// TIA Portal project "Nastro con lavorazione HMI_lab" (V16)

(* hardware
DEVICE "HMI_1"  KTP700 Basic PN
   slot 0: "HMI_1"  KTP700 Basic PN  6AV2 123-2GB03-0AX0  16.0.0.0
   slot 1: "HMI_RT_1"  KTP700 Basic PN  6AV2 123-2GB03-0AX0  16.0.0.0
   slot 5: "HMI_1.IE_CP_1"  PROFINET Interface  16.0.0.0
      slot 1: "Interfaccia_1 PROFINET"  PROFINET Interface
         slot 1: "Porta_1"  Port
DEVICE "S7-1200 station_1"  S7-1200 Station
   slot 0: "Telaio di montaggio_0"  S7-1200 Rack  Rack  V1.0
   slot 1: "PLC_1"  CPU 1215C DC/DC/Rly  6ES7 215-1HG40-0XB0  V4.2
*)

// ===== PLC "PLC_1"  CPU 1215C DC/DC/Rly =====

VAR_GLOBAL   // PLC tag table "Tabella delle variabili standard"
   "Passo_0" AT %M0.0 : Bool;
   "Passo_1" AT %M0.1 : Bool;
   "Passo_2" AT %M0.2 : Bool;
   "Passo_3" AT %M0.3 : Bool;
   "Passo_4" AT %M0.4 : Bool;
   "BC_inizio" AT %I0.0 : Bool;
   "BC_fine" AT %I0.1 : Bool;
   "SQ_alto" AT %I0.2 : Bool;
   "SB_basso" AT %I0.3 : Bool;
   "Avanti nastro" AT %Q0.0 : Bool;
   "Indietro nastro" AT %Q0.1 : Bool;
   "Passo_5" AT %M0.5 : Bool;
   "Discesa lavorazione" AT %Q0.2 : Bool;
   "Salita lavorazione" AT %Q0.3 : Bool;
   "Clock_Byte" AT %MB10 : Byte;
   "Clock_10Hz" AT %M10.0 : Bool;
   "Clock_5Hz" AT %M10.1 : Bool;
   "Clock_2.5Hz" AT %M10.2 : Bool;
   "Clock_2Hz" AT %M10.3 : Bool;
   "Clock_1.25Hz" AT %M10.4 : Bool;
   "Clock_1Hz" AT %M10.5 : Bool;
   "Clock_0.625Hz" AT %M10.6 : Bool;
   "Clock_0.5Hz" AT %M10.7 : Bool;
END_VAR

DATA_BLOCK "Blocco_dati_HMI"   // DB1
{ S7_Optimized_Access := 'TRUE' }
VERSION : 0.1
   VAR
      jog_start : Bool;
      jog_BC_inizio : Bool;
      M_cicli : Bool;
      "movimento cilindretto" : Int;
      M_clock_veloce : Bool;
      M_clock_lento : Bool;
      "movimento lavorazione" : Int;
      jog_emergenza : Bool;
      jog_ripristino : Bool;
      M_tempo_lav : Bool;
      jog_BC_fine : Bool;
      jog_SQ_basso : Bool;
      jog_SQ_alto : Bool;
      preset_tempo_lav : Time;
      jog_carica_impostazioni : Bool;
      imposta_tempo_lav : Time;
      "lettura tempo_lav" : Time;
      "imposta numero di cicli" : Int;
      "lettura numero di cicli" : Int;
      preset_conteggio_cicli : Int;
      M_ripristino_cilindretto : Bool;
      M_ripristino_lav : Bool;
      Spia_BC_inizio : Bool;
      Spia_BC_fine : Bool;
      Spia_SQ_alto : Bool;
      "Spia _SQ_basso" : Bool;
      "Spia organi in movimento" : Bool;
      M_ripristino_lav_reale : Bool;
      M_ripristino_cilindro_reale_1 : Bool;
   END_VAR
BEGIN
END_DATA_BLOCK

// folder: System blocks/Program resources

DATA_BLOCK "Clock_lento"   // DB2
{ S7_Optimized_Access := 'TRUE' }
AUTHOR : Simatic
FAMILY : IEC
NAME : IEC_TMR
VERSION : 1.0
// stored: InstanceOfName IEC_TIMER
"IEC_TIMER"
BEGIN
END_DATA_BLOCK

DATA_BLOCK "Clock_veloce"   // DB3
{ S7_Optimized_Access := 'TRUE' }
AUTHOR : Simatic
FAMILY : IEC
NAME : IEC_TMR
VERSION : 1.0
// stored: InstanceOfName IEC_TIMER
"IEC_TIMER"
BEGIN
END_DATA_BLOCK

DATA_BLOCK "Tempo_lav"   // DB4
{ S7_Optimized_Access := 'TRUE' }
AUTHOR : Simatic
FAMILY : IEC
NAME : IEC_TMR
VERSION : 1.0
// stored: InstanceOfName IEC_TIMER
"IEC_TIMER"
BEGIN
END_DATA_BLOCK

DATA_BLOCK "Conteggio cicli"   // DB5
{ S7_Optimized_Access := 'TRUE' }
AUTHOR : Simatic
FAMILY : IEC
NAME : CNTR
VERSION : 1.0
// stored: InstanceOfName IEC_COUNTER
"IEC_COUNTER"
BEGIN
END_DATA_BLOCK

// folder: (top level)

FUNCTION "Ripristino" : Void   // FC1, LAD
{ S7_Optimized_Access := 'TRUE' }
VERSION : 0.1
BEGIN

REGION Network 1
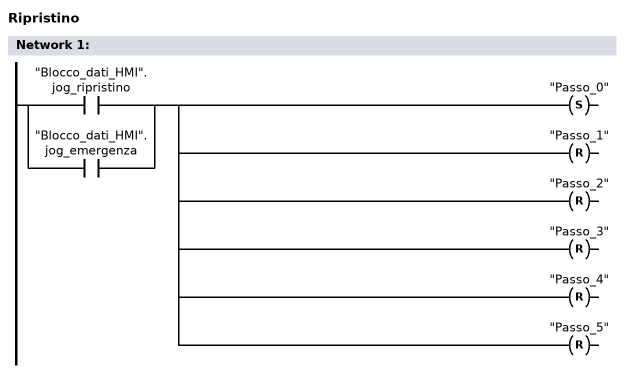
   RUNG wire#powerrail
      Contact( "Blocco_dati_HMI".jog_ripristino )
      wire#w1
      S_Coil( "Passo_0" )
   END_RUNG
   RUNG wire#powerrail
      Contact( "Blocco_dati_HMI".jog_emergenza )
   END_RUNG wire#w1
   RUNG wire#w1
      R_Coil( "Passo_1" )
   END_RUNG
   RUNG wire#w1
      R_Coil( "Passo_2" )
   END_RUNG
   RUNG wire#w1
      R_Coil( "Passo_3" )
   END_RUNG
   RUNG wire#w1
      R_Coil( "Passo_4" )
   END_RUNG
   RUNG wire#w1
      R_Coil( "Passo_5" )
   END_RUNG
   // the same network as SCL:
   IF "Blocco_dati_HMI".jog_ripristino OR "Blocco_dati_HMI".jog_emergenza THEN
       "Passo_0" := TRUE;
       "Passo_1" := FALSE;
       "Passo_2" := FALSE;
       "Passo_3" := FALSE;
       "Passo_4" := FALSE;
       "Passo_5" := FALSE;
   END_IF;
END_REGION
END_FUNCTION

FUNCTION "Struttura dei passi" : Void   // FC2, LAD
{ S7_Optimized_Access := 'TRUE' }
VERSION : 0.1
   VAR_TEMP   // added for the SCL form of the ladder/FBD networks
      _w1 : Bool;
   END_VAR
BEGIN

REGION Network 1
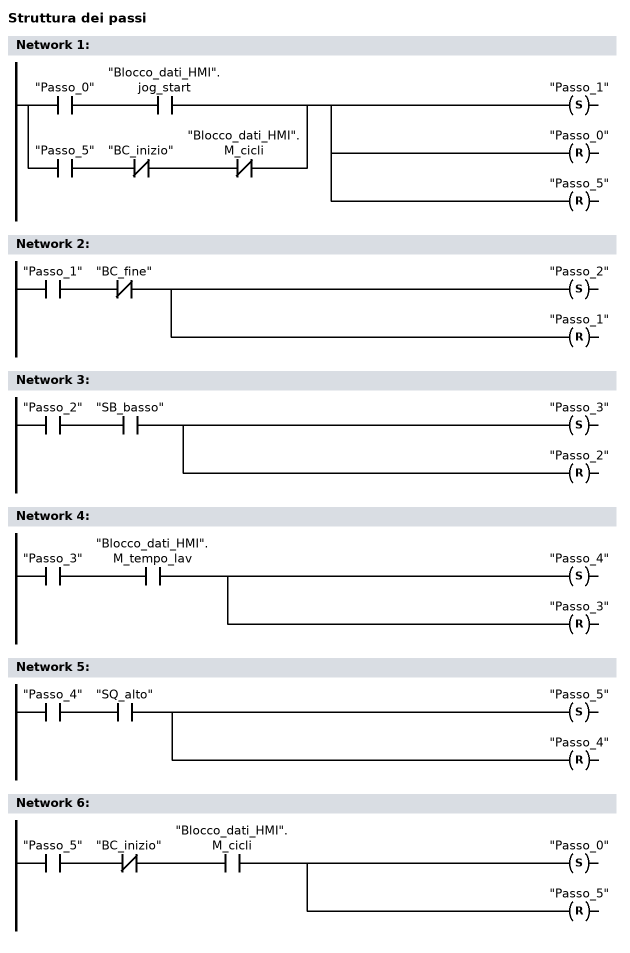
   RUNG wire#powerrail
      Contact( "Passo_0" )
      Contact( "Blocco_dati_HMI".jog_start )
      wire#w1
      S_Coil( "Passo_1" )
   END_RUNG
   RUNG wire#powerrail
      Contact( "Passo_5" )
      I_Contact( "BC_inizio" )
      I_Contact( "Blocco_dati_HMI".M_cicli )
   END_RUNG wire#w1
   RUNG wire#w1
      R_Coil( "Passo_0" )
   END_RUNG
   RUNG wire#w1
      R_Coil( "Passo_5" )
   END_RUNG
   // the same network as SCL:
   IF ("Passo_0" AND "Blocco_dati_HMI".jog_start) OR ("Passo_5" AND NOT "BC_inizio" AND NOT "Blocco_dati_HMI".M_cicli) THEN
       "Passo_1" := TRUE;
   END_IF;
   #_w1 := ("Passo_0" AND "Blocco_dati_HMI".jog_start) OR ("Passo_5" AND NOT "BC_inizio" AND NOT "Blocco_dati_HMI".M_cicli);
   IF #_w1 THEN
       "Passo_0" := FALSE;
       "Passo_5" := FALSE;
   END_IF;
END_REGION

REGION Network 2
   RUNG wire#powerrail
      Contact( "Passo_1" )
      I_Contact( "BC_fine" )
      wire#w1
      S_Coil( "Passo_2" )
   END_RUNG
   RUNG wire#w1
      R_Coil( "Passo_1" )
   END_RUNG
   // the same network as SCL:
   IF "Passo_1" AND NOT "BC_fine" THEN
       "Passo_2" := TRUE;
       "Passo_1" := FALSE;
   END_IF;
END_REGION

REGION Network 3
   RUNG wire#powerrail
      Contact( "Passo_2" )
      Contact( "SB_basso" )
      wire#w1
      S_Coil( "Passo_3" )
   END_RUNG
   RUNG wire#w1
      R_Coil( "Passo_2" )
   END_RUNG
   // the same network as SCL:
   IF "Passo_2" AND "SB_basso" THEN
       "Passo_3" := TRUE;
       "Passo_2" := FALSE;
   END_IF;
END_REGION

REGION Network 4
   RUNG wire#powerrail
      Contact( "Passo_3" )
      Contact( "Blocco_dati_HMI".M_tempo_lav )
      wire#w1
      S_Coil( "Passo_4" )
   END_RUNG
   RUNG wire#w1
      R_Coil( "Passo_3" )
   END_RUNG
   // the same network as SCL:
   IF "Passo_3" AND "Blocco_dati_HMI".M_tempo_lav THEN
       "Passo_4" := TRUE;
       "Passo_3" := FALSE;
   END_IF;
END_REGION

REGION Network 5
   RUNG wire#powerrail
      Contact( "Passo_4" )
      Contact( "SQ_alto" )
      wire#w1
      S_Coil( "Passo_5" )
   END_RUNG
   RUNG wire#w1
      R_Coil( "Passo_4" )
   END_RUNG
   // the same network as SCL:
   IF "Passo_4" AND "SQ_alto" THEN
       "Passo_5" := TRUE;
       "Passo_4" := FALSE;
   END_IF;
END_REGION

REGION Network 6
   RUNG wire#powerrail
      Contact( "Passo_5" )
      I_Contact( "BC_inizio" )
      Contact( "Blocco_dati_HMI".M_cicli )
      wire#w1
      S_Coil( "Passo_0" )
   END_RUNG
   RUNG wire#w1
      R_Coil( "Passo_5" )
   END_RUNG
   // the same network as SCL:
   IF "Passo_5" AND NOT "BC_inizio" AND "Blocco_dati_HMI".M_cicli THEN
       "Passo_0" := TRUE;
       "Passo_5" := FALSE;
   END_IF;
END_REGION
END_FUNCTION

FUNCTION "Attivazione delle uscite" : Void   // FC3, LAD
{ S7_Optimized_Access := 'TRUE' }
VERSION : 0.1
BEGIN

REGION Network 1
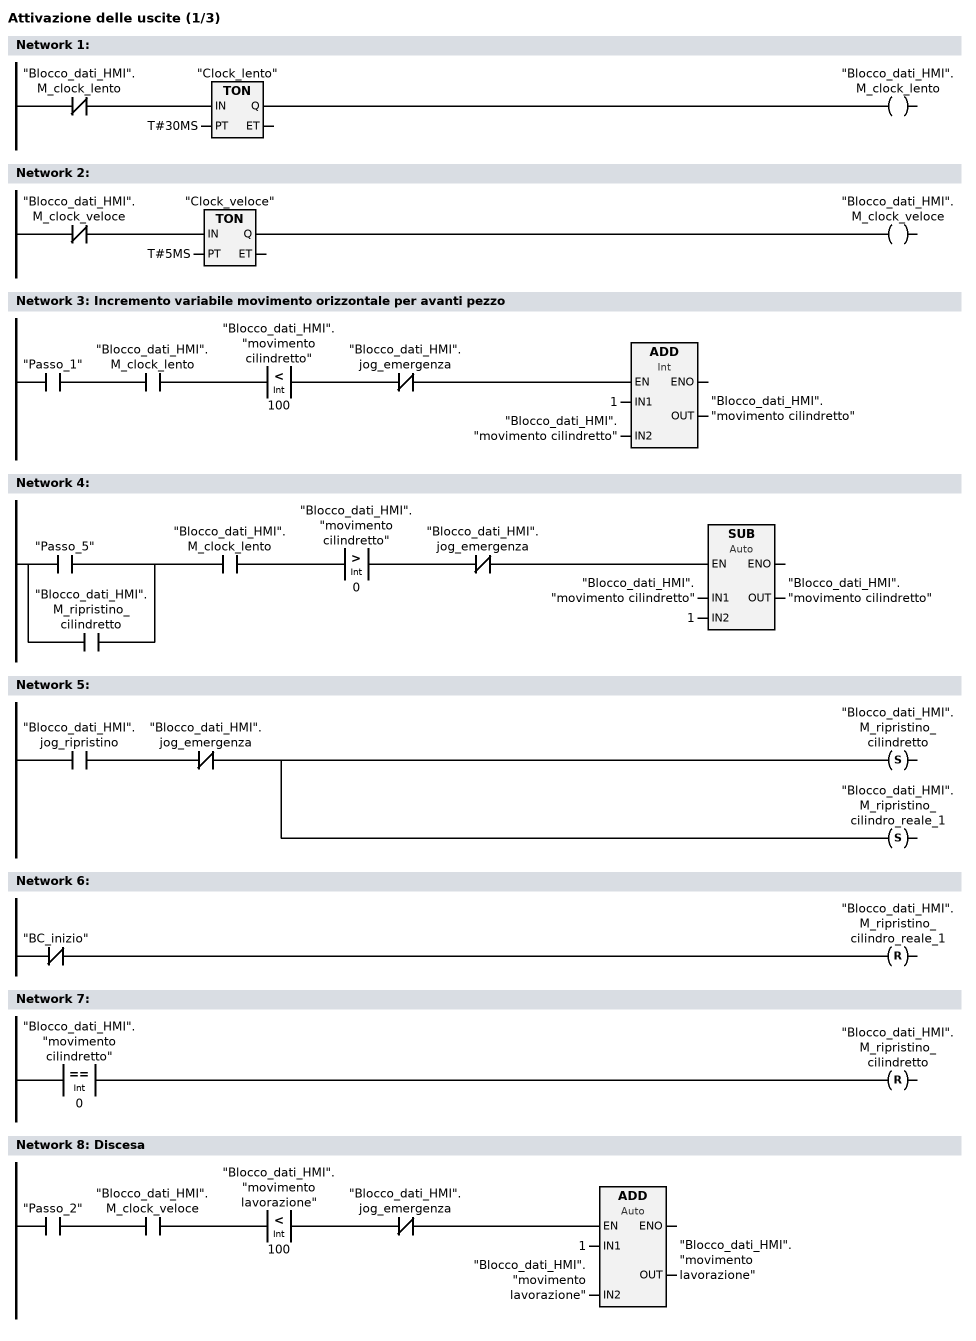
   "Clock_lento".TON(IN := NOT "Blocco_dati_HMI".M_clock_lento, PT := T#30MS);
   "Blocco_dati_HMI".M_clock_lento := "Clock_lento".Q;
END_REGION

REGION Network 2
   "Clock_veloce".TON(IN := NOT "Blocco_dati_HMI".M_clock_veloce, PT := T#5MS);
   "Blocco_dati_HMI".M_clock_veloce := "Clock_veloce".Q;
END_REGION

REGION Network 3: Incremento variabile movimento orizzontale per avanti pezzo
   RUNG wire#powerrail
      Contact( "Passo_1" )
      Contact( "Blocco_dati_HMI".M_clock_lento )
      { S7_Templates := "SrcType := Int" } LT_Contact(in1 := "Blocco_dati_HMI"."movimento cilindretto", in2 := 100)
      I_Contact( "Blocco_dati_HMI".jog_emergenza )
      { S7_Templates := "SrcType := Int" } Add(in1 := 1, in2 := "Blocco_dati_HMI"."movimento cilindretto", out => "Blocco_dati_HMI"."movimento cilindretto")
   END_RUNG
   // the same network as SCL:
   IF "Passo_1" AND "Blocco_dati_HMI".M_clock_lento AND ("Blocco_dati_HMI"."movimento cilindretto" < 100) AND NOT "Blocco_dati_HMI".jog_emergenza THEN
       "Blocco_dati_HMI"."movimento cilindretto" := 1 + "Blocco_dati_HMI"."movimento cilindretto";
   END_IF;
END_REGION

REGION Network 4
   RUNG wire#powerrail
      Contact( "Passo_5" )
      wire#w1
      Contact( "Blocco_dati_HMI".M_clock_lento )
      { S7_Templates := "SrcType := Int" } GT_Contact(in1 := "Blocco_dati_HMI"."movimento cilindretto", in2 := 0)
      I_Contact( "Blocco_dati_HMI".jog_emergenza )
      Sub(in1 := "Blocco_dati_HMI"."movimento cilindretto", in2 := 1, out => "Blocco_dati_HMI"."movimento cilindretto")
   END_RUNG
   RUNG wire#powerrail
      Contact( "Blocco_dati_HMI".M_ripristino_cilindretto )
   END_RUNG wire#w1
   // the same network as SCL:
   IF ("Passo_5" OR "Blocco_dati_HMI".M_ripristino_cilindretto) AND "Blocco_dati_HMI".M_clock_lento AND ("Blocco_dati_HMI"."movimento cilindretto" > 0) AND NOT "Blocco_dati_HMI".jog_emergenza THEN
       "Blocco_dati_HMI"."movimento cilindretto" := "Blocco_dati_HMI"."movimento cilindretto" - 1;
   END_IF;
END_REGION

REGION Network 5
   RUNG wire#powerrail
      Contact( "Blocco_dati_HMI".jog_ripristino )
      I_Contact( "Blocco_dati_HMI".jog_emergenza )
      wire#w1
      S_Coil( "Blocco_dati_HMI".M_ripristino_cilindretto )
   END_RUNG
   RUNG wire#w1
      S_Coil( "Blocco_dati_HMI".M_ripristino_cilindro_reale_1 )
   END_RUNG
   // the same network as SCL:
   IF "Blocco_dati_HMI".jog_ripristino AND NOT "Blocco_dati_HMI".jog_emergenza THEN
       "Blocco_dati_HMI".M_ripristino_cilindretto := TRUE;
       "Blocco_dati_HMI".M_ripristino_cilindro_reale_1 := TRUE;
   END_IF;
END_REGION

REGION Network 6
   RUNG wire#powerrail
      I_Contact( "BC_inizio" )
      R_Coil( "Blocco_dati_HMI".M_ripristino_cilindro_reale_1 )
   END_RUNG
   // the same network as SCL:
   IF NOT "BC_inizio" THEN "Blocco_dati_HMI".M_ripristino_cilindro_reale_1 := FALSE; END_IF;
END_REGION

REGION Network 7
   RUNG wire#powerrail
      { S7_Templates := "SrcType := Int" } EQ_Contact(in1 := "Blocco_dati_HMI"."movimento cilindretto", in2 := 0)
      R_Coil( "Blocco_dati_HMI".M_ripristino_cilindretto )
   END_RUNG
   // the same network as SCL:
   IF "Blocco_dati_HMI"."movimento cilindretto" = 0 THEN
       "Blocco_dati_HMI".M_ripristino_cilindretto := FALSE;
   END_IF;
END_REGION

REGION Network 8: Discesa
   RUNG wire#powerrail
      Contact( "Passo_2" )
      Contact( "Blocco_dati_HMI".M_clock_veloce )
      { S7_Templates := "SrcType := Int" } LT_Contact(in1 := "Blocco_dati_HMI"."movimento lavorazione", in2 := 100)
      I_Contact( "Blocco_dati_HMI".jog_emergenza )
      Add(in1 := 1, in2 := "Blocco_dati_HMI"."movimento lavorazione", out => "Blocco_dati_HMI"."movimento lavorazione")
   END_RUNG
   // the same network as SCL:
   IF "Passo_2" AND "Blocco_dati_HMI".M_clock_veloce AND ("Blocco_dati_HMI"."movimento lavorazione" < 100) AND NOT "Blocco_dati_HMI".jog_emergenza THEN
       "Blocco_dati_HMI"."movimento lavorazione" := 1 + "Blocco_dati_HMI"."movimento lavorazione";
   END_IF;
END_REGION

REGION Network 9: salita
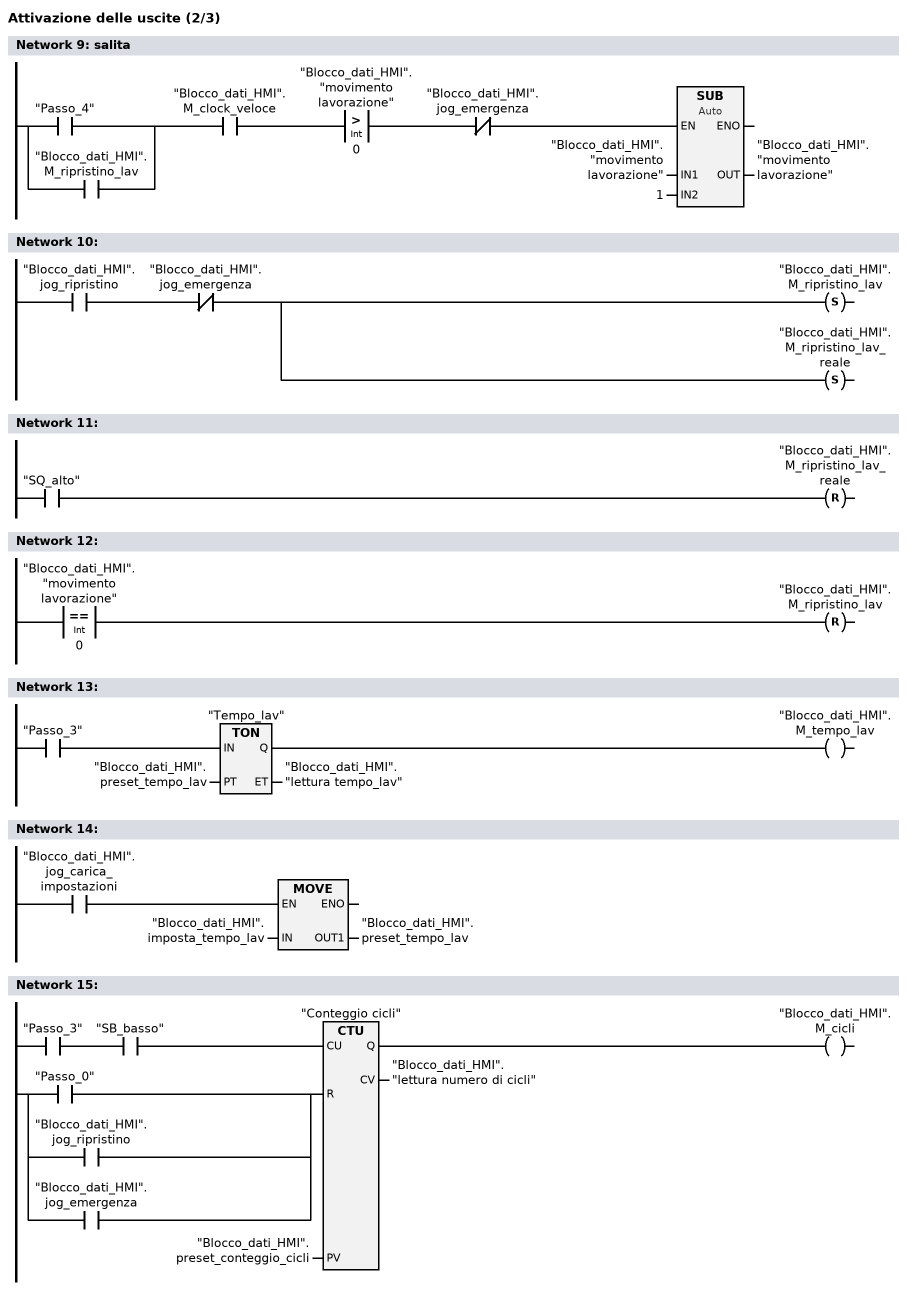
   RUNG wire#powerrail
      Contact( "Passo_4" )
      wire#w1
      Contact( "Blocco_dati_HMI".M_clock_veloce )
      { S7_Templates := "SrcType := Int" } GT_Contact(in1 := "Blocco_dati_HMI"."movimento lavorazione", in2 := 0)
      I_Contact( "Blocco_dati_HMI".jog_emergenza )
      Sub(in1 := "Blocco_dati_HMI"."movimento lavorazione", in2 := 1, out => "Blocco_dati_HMI"."movimento lavorazione")
   END_RUNG
   RUNG wire#powerrail
      Contact( "Blocco_dati_HMI".M_ripristino_lav )
   END_RUNG wire#w1
   // the same network as SCL:
   IF ("Passo_4" OR "Blocco_dati_HMI".M_ripristino_lav) AND "Blocco_dati_HMI".M_clock_veloce AND ("Blocco_dati_HMI"."movimento lavorazione" > 0) AND NOT "Blocco_dati_HMI".jog_emergenza THEN
       "Blocco_dati_HMI"."movimento lavorazione" := "Blocco_dati_HMI"."movimento lavorazione" - 1;
   END_IF;
END_REGION

REGION Network 10
   RUNG wire#powerrail
      Contact( "Blocco_dati_HMI".jog_ripristino )
      I_Contact( "Blocco_dati_HMI".jog_emergenza )
      wire#w1
      S_Coil( "Blocco_dati_HMI".M_ripristino_lav )
   END_RUNG
   RUNG wire#w1
      S_Coil( "Blocco_dati_HMI".M_ripristino_lav_reale )
   END_RUNG
   // the same network as SCL:
   IF "Blocco_dati_HMI".jog_ripristino AND NOT "Blocco_dati_HMI".jog_emergenza THEN
       "Blocco_dati_HMI".M_ripristino_lav := TRUE;
       "Blocco_dati_HMI".M_ripristino_lav_reale := TRUE;
   END_IF;
END_REGION

REGION Network 11
   RUNG wire#powerrail
      Contact( "SQ_alto" )
      R_Coil( "Blocco_dati_HMI".M_ripristino_lav_reale )
   END_RUNG
   // the same network as SCL:
   IF "SQ_alto" THEN "Blocco_dati_HMI".M_ripristino_lav_reale := FALSE; END_IF;
END_REGION

REGION Network 12
   RUNG wire#powerrail
      { S7_Templates := "SrcType := Int" } EQ_Contact(in1 := "Blocco_dati_HMI"."movimento lavorazione", in2 := 0)
      R_Coil( "Blocco_dati_HMI".M_ripristino_lav )
   END_RUNG
   // the same network as SCL:
   IF "Blocco_dati_HMI"."movimento lavorazione" = 0 THEN "Blocco_dati_HMI".M_ripristino_lav := FALSE; END_IF;
END_REGION

REGION Network 13
   "Tempo_lav".TON(IN := "Passo_3",
                   PT := "Blocco_dati_HMI".preset_tempo_lav,
                   ET => "Blocco_dati_HMI"."lettura tempo_lav");
   "Blocco_dati_HMI".M_tempo_lav := "Tempo_lav".Q;
END_REGION

REGION Network 14
   RUNG wire#powerrail
      Contact( "Blocco_dati_HMI".jog_carica_impostazioni )
      Move(in := "Blocco_dati_HMI".imposta_tempo_lav, out1 => "Blocco_dati_HMI".preset_tempo_lav)
   END_RUNG
   // the same network as SCL:
   IF "Blocco_dati_HMI".jog_carica_impostazioni THEN
       "Blocco_dati_HMI".preset_tempo_lav := "Blocco_dati_HMI".imposta_tempo_lav;
   END_IF;
END_REGION

REGION Network 15
   "Conteggio cicli".CTU(CU := "Passo_3" AND "SB_basso",
                         R := "Passo_0" OR "Blocco_dati_HMI".jog_ripristino OR "Blocco_dati_HMI".jog_emergenza,
                         PV := "Blocco_dati_HMI".preset_conteggio_cicli,
                         CV => "Blocco_dati_HMI"."lettura numero di cicli");
   "Blocco_dati_HMI".M_cicli := "Conteggio cicli".Q;
END_REGION

REGION Network 16
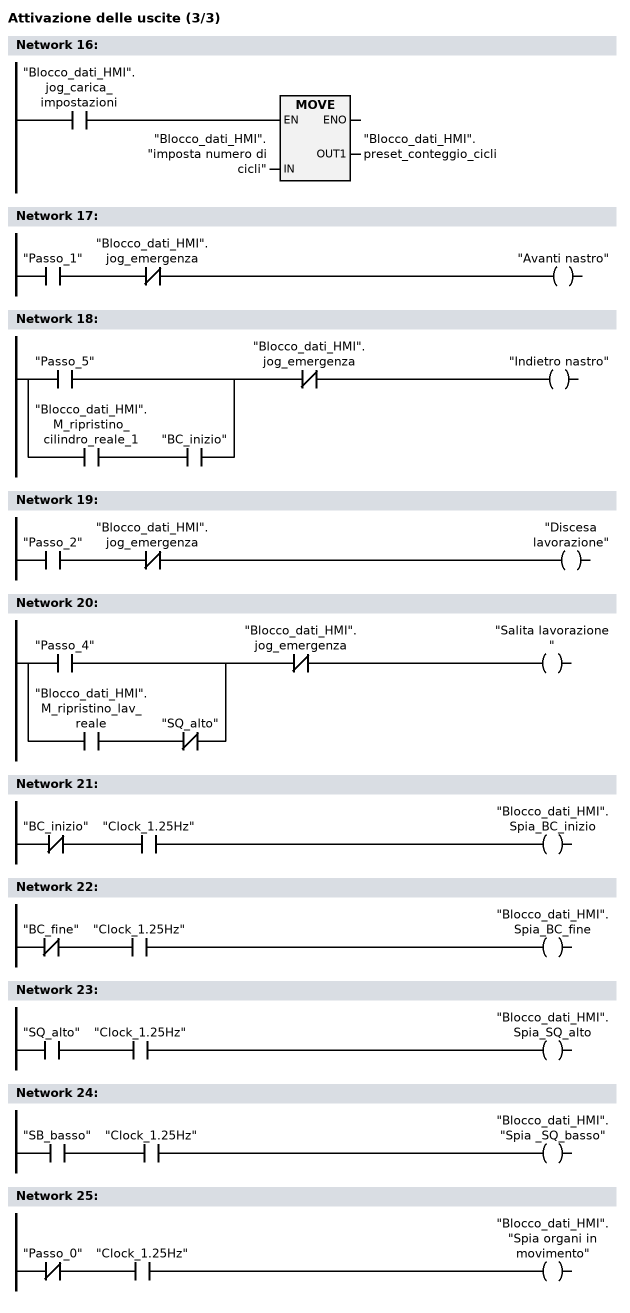
   RUNG wire#powerrail
      Contact( "Blocco_dati_HMI".jog_carica_impostazioni )
      Move(in := "Blocco_dati_HMI"."imposta numero di cicli", out1 => "Blocco_dati_HMI".preset_conteggio_cicli)
   END_RUNG
   // the same network as SCL:
   IF "Blocco_dati_HMI".jog_carica_impostazioni THEN
       "Blocco_dati_HMI".preset_conteggio_cicli := "Blocco_dati_HMI"."imposta numero di cicli";
   END_IF;
END_REGION

REGION Network 17
   RUNG wire#powerrail
      Contact( "Passo_1" )
      I_Contact( "Blocco_dati_HMI".jog_emergenza )
      Coil( "Avanti nastro" )
   END_RUNG
   // the same network as SCL:
   "Avanti nastro" := "Passo_1" AND NOT "Blocco_dati_HMI".jog_emergenza;
END_REGION

REGION Network 18
   RUNG wire#powerrail
      Contact( "Passo_5" )
      wire#w1
      I_Contact( "Blocco_dati_HMI".jog_emergenza )
      Coil( "Indietro nastro" )
   END_RUNG
   RUNG wire#powerrail
      Contact( "Blocco_dati_HMI".M_ripristino_cilindro_reale_1 )
      Contact( "BC_inizio" )
   END_RUNG wire#w1
   // the same network as SCL:
   "Indietro nastro" := ("Passo_5" OR ("Blocco_dati_HMI".M_ripristino_cilindro_reale_1 AND "BC_inizio")) AND NOT "Blocco_dati_HMI".jog_emergenza;
END_REGION

REGION Network 19
   RUNG wire#powerrail
      Contact( "Passo_2" )
      I_Contact( "Blocco_dati_HMI".jog_emergenza )
      Coil( "Discesa lavorazione" )
   END_RUNG
   // the same network as SCL:
   "Discesa lavorazione" := "Passo_2" AND NOT "Blocco_dati_HMI".jog_emergenza;
END_REGION

REGION Network 20
   RUNG wire#powerrail
      Contact( "Passo_4" )
      wire#w1
      I_Contact( "Blocco_dati_HMI".jog_emergenza )
      Coil( "Salita lavorazione" )
   END_RUNG
   RUNG wire#powerrail
      Contact( "Blocco_dati_HMI".M_ripristino_lav_reale )
      I_Contact( "SQ_alto" )
   END_RUNG wire#w1
   // the same network as SCL:
   "Salita lavorazione" := ("Passo_4" OR ("Blocco_dati_HMI".M_ripristino_lav_reale AND NOT "SQ_alto")) AND NOT "Blocco_dati_HMI".jog_emergenza;
END_REGION

REGION Network 21
   RUNG wire#powerrail
      I_Contact( "BC_inizio" )
      Contact( "Clock_1.25Hz" )
      Coil( "Blocco_dati_HMI".Spia_BC_inizio )
   END_RUNG
   // the same network as SCL:
   "Blocco_dati_HMI".Spia_BC_inizio := NOT "BC_inizio" AND "Clock_1.25Hz";
END_REGION

REGION Network 22
   RUNG wire#powerrail
      I_Contact( "BC_fine" )
      Contact( "Clock_1.25Hz" )
      Coil( "Blocco_dati_HMI".Spia_BC_fine )
   END_RUNG
   // the same network as SCL:
   "Blocco_dati_HMI".Spia_BC_fine := NOT "BC_fine" AND "Clock_1.25Hz";
END_REGION

REGION Network 23
   RUNG wire#powerrail
      Contact( "SQ_alto" )
      Contact( "Clock_1.25Hz" )
      Coil( "Blocco_dati_HMI".Spia_SQ_alto )
   END_RUNG
   // the same network as SCL:
   "Blocco_dati_HMI".Spia_SQ_alto := "SQ_alto" AND "Clock_1.25Hz";
END_REGION

REGION Network 24
   RUNG wire#powerrail
      Contact( "SB_basso" )
      Contact( "Clock_1.25Hz" )
      Coil( "Blocco_dati_HMI"."Spia _SQ_basso" )
   END_RUNG
   // the same network as SCL:
   "Blocco_dati_HMI"."Spia _SQ_basso" := "SB_basso" AND "Clock_1.25Hz";
END_REGION

REGION Network 25
   RUNG wire#powerrail
      I_Contact( "Passo_0" )
      Contact( "Clock_1.25Hz" )
      Coil( "Blocco_dati_HMI"."Spia organi in movimento" )
   END_RUNG
   // the same network as SCL:
   "Blocco_dati_HMI"."Spia organi in movimento" := NOT "Passo_0" AND "Clock_1.25Hz";
END_REGION
END_FUNCTION

ORGANIZATION_BLOCK "Main"   // OB1, LAD, ProgramCycle
TITLE = "Main Program Sweep (Cycle)"
{ S7_Optimized_Access := 'TRUE' }
VERSION : 0.1
   VAR_INPUT
      Initial_Call : Bool;   // Initial call of this OB
      Remanence : Bool;   // =True, if remanent data are available
   END_VAR
BEGIN

REGION Network 1
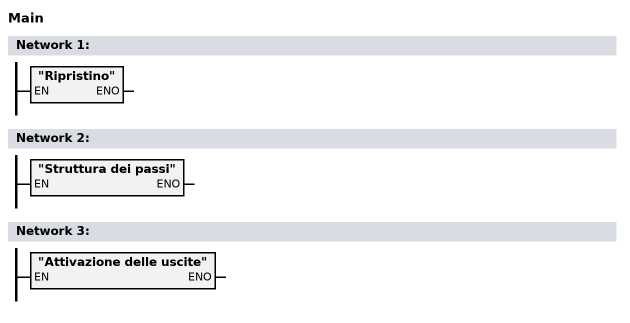
   RUNG wire#powerrail
      "Ripristino"()
   END_RUNG
   // the same network as SCL:
   "Ripristino"();
END_REGION

REGION Network 2
   RUNG wire#powerrail
      "Struttura dei passi"()
   END_RUNG
   // the same network as SCL:
   "Struttura dei passi"();
END_REGION

REGION Network 3
   RUNG wire#powerrail
      "Attivazione delle uscite"()
   END_RUNG
   // the same network as SCL:
   "Attivazione delle uscite"();
END_REGION
END_ORGANIZATION_BLOCK

(* ===== HMI "HMI_RT_1" =====
system functions are stored by id; their names below are inferred from use
connection "HMI_Collegamento_1": ETHERNET, SMART_S7_1200_OMS

HMI tags "Tabella delle variabili standard"
   "Blocco_dati_HMI_jog_emergenza" : Bool = PLC Blocco_dati_HMI.jog_emergenza, 100 ms
   "Blocco_dati_HMI_jog_ripristino" : Bool = PLC Blocco_dati_HMI.jog_ripristino, 100 ms
   "Blocco_dati_HMI_jog_start" : Bool = PLC Blocco_dati_HMI.jog_start, 100 ms
   "Blocco_dati_HMI_imposta_tempo_lav" : Time = PLC Blocco_dati_HMI.imposta_tempo_lav, 100 ms
   "Blocco_dati_HMI_preset_tempo_lav" : Time = PLC Blocco_dati_HMI.preset_tempo_lav, 100 ms
   "Blocco_dati_HMI_lettura tempo_lav" : Time = PLC Blocco_dati_HMI."lettura tempo_lav", 100 ms
   "Blocco_dati_HMI_imposta numero di cicli" : Int = PLC Blocco_dati_HMI."imposta numero di cicli", 100 ms
   "Blocco_dati_HMI_preset_conteggio_cicli" : Int = PLC Blocco_dati_HMI.preset_conteggio_cicli, 100 ms
   "Blocco_dati_HMI_lettura numero di cicli" : Int = PLC Blocco_dati_HMI."lettura numero di cicli", 100 ms
   "Blocco_dati_HMI_jog_carica_impostazioni" : Bool = PLC Blocco_dati_HMI.jog_carica_impostazioni, 100 ms
   "Blocco_dati_HMI_jog_BC_inizio" : Bool = PLC Blocco_dati_HMI.jog_BC_inizio, 100 ms
   "Blocco_dati_HMI_jog_BC_fine" : Bool = PLC Blocco_dati_HMI.jog_BC_fine, 100 ms
   "Blocco_dati_HMI_jog_SQ_basso" : Bool = PLC Blocco_dati_HMI.jog_SQ_basso, 100 ms
   "Blocco_dati_HMI_jog_SQ_alto" : Bool = PLC Blocco_dati_HMI.jog_SQ_alto, 100 ms
   "Blocco_dati_HMI_movimento cilindretto" : Int = PLC Blocco_dati_HMI."movimento cilindretto", 100 ms
   "Blocco_dati_HMI_movimento lavorazione" : Int = PLC Blocco_dati_HMI."movimento lavorazione", 100 ms
   "Blocco_dati_HMI_Spia organi in movimento" : Bool = PLC Blocco_dati_HMI."Spia organi in movimento", 100 ms
   "Blocco_dati_HMI_Spia_SQ_alto" : Bool = PLC Blocco_dati_HMI.Spia_SQ_alto, 100 ms
   "Blocco_dati_HMI_Spia _SQ_basso" : Bool = PLC Blocco_dati_HMI."Spia _SQ_basso", 100 ms
   "Blocco_dati_HMI_Spia_BC_fine" : Bool = PLC Blocco_dati_HMI.Spia_BC_fine, 100 ms
   "Blocco_dati_HMI_Spia_BC_inizio" : Bool = PLC Blocco_dati_HMI.Spia_BC_inizio, 100 ms

screen "Pagina_1" 800x480
   Softkey "Softkey_F1" at 0,0 size 0x0
      on KeyDown: ActivateScreen("Pagina_1", 0)
   Softkey "Softkey_F2" at 0,0 size 0x0
      on KeyDown: ActivateScreen("Pagina_2", 0)

screen "Pagina_2" 800x480
   Softkey "Softkey_F1" at 0,0 size 0x0
      on KeyDown: ActivateScreen("Pagina_1", 0)
   Softkey "Softkey_F2" at 0,0 size 0x0
      on KeyDown: ActivateScreen("Pagina_2", 0)
   Rectangle "Rettangolo_2" at 526,291 size 46x43
      HorizontalMovement <- "Blocco_dati_HMI_movimento cilindretto"
   Switch "Pushbutton_Emergency" at 53,43 size 80x80; CaptionText 'Switch'; TextOff '0'; TextOn '1'; PictureOff "Pushbutton_Emergency_Off_256c"; PictureOn "Pushbutton_Emergency_On_256c"
      on SwitchOn: SetBit("Blocco_dati_HMI_jog_emergenza")
      on SwitchOff: ResetBit("Blocco_dati_HMI_jog_emergenza")
   Button "FB_Home_Round" at 211,48 size 50x50; TextOff 'Text'; PictureOn "FB_Home_Round_Pressed_256c"; PictureOff "FB_Home_Round_Released_256c"
      on Press: SetBit("Blocco_dati_HMI_jog_ripristino")
      on Release: ResetBit("Blocco_dati_HMI_jog_ripristino")
   Button "FB_Right_Round" at 318,48 size 50x50; TextOff 'Text'; PictureOn "FB_Right_Round_Pressed_256c"; PictureOff "FB_Right_Round_Released_256c"
      on Press: SetBit("Blocco_dati_HMI_jog_start")
      on Release: ResetBit("Blocco_dati_HMI_jog_start")
   IOField "Campo I/O_1" at 47,240 size 58x32; FormatPattern 9999
      ProcessValue <- "Blocco_dati_HMI_imposta_tempo_lav"
   IOField "Campo I/O_2" at 47,403 size 58x32; FormatPattern 9999
      ProcessValue <- "Blocco_dati_HMI_imposta numero di cicli"
   IOField "Campo I/O_3" at 183,240 size 58x32; FormatPattern 9999
      ProcessValue <- "Blocco_dati_HMI_preset_tempo_lav"
   IOField "Campo I/O_4" at 183,403 size 58x32; FormatPattern 9999
      ProcessValue <- "Blocco_dati_HMI_preset_conteggio_cicli"
   IOField "Campo I/O_5" at 321,240 size 58x32; FormatPattern 9999
      ProcessValue <- "Blocco_dati_HMI_lettura tempo_lav"
   IOField "Campo I/O_6" at 320,402 size 58x32; FormatPattern 9999
      ProcessValue <- "Blocco_dati_HMI_lettura numero di cicli"
   Button "FB_Plus_Round" at 116,310 size 50x50; TextOff 'Text'; PictureOn "FB_Plus_Round_Pressed_256c"; PictureOff "FB_Plus_Round_Released_256c"
      on Press: SetBit("Blocco_dati_HMI_jog_carica_impostazioni")
      on Release: ResetBit("Blocco_dati_HMI_jog_carica_impostazioni")
   TextField "Casella di testo_1" at 53,19 size 76x20; Text 'Emergenza'
   TextField "Casella di testo_2" at 212,19 size 41x20; Text 'Home'
   TextField "Casella di testo_3" at 488,48 size 65x20; Text 'Macchina'
   TextField "Casella di testo_5" at 42,201 size 87x20; Text 'Digita tempo'
   TextField "Casella di testo_6" at 42,216 size 80x20; Text 'lavorazione'
   TextField "Casella di testo_4" at 183,201 size 47x20; Text 'Tempo'
   TextField "Casella di testo_7" at 183,216 size 80x20; Text 'lavorazione'
   TextField "Casella di testo_8" at 316,201 size 68x20; Text 'Visualizza'
   TextField "Casella di testo_9" at 316,216 size 88x20; Text 'tempo di lav.'
   TextField "Casella di testo_10" at 103,275 size 45x20; Text 'Carica'
   TextField "Casella di testo_11" at 103,290 size 85x20; Text 'impostazioni'
   TextField "Casella di testo_12" at 42,367 size 95x20; Text 'Digita numero'
   TextField "Casella di testo_13" at 42,382 size 43x20; Text 'di cicli'
   TextField "Casella di testo_14" at 184,368 size 58x20; Text 'Numero'
   TextField "Casella di testo_15" at 184,383 size 43x20; Text 'di cicli'
   TextField "Casella di testo_16" at 321,367 size 68x20; Text 'Visualizza'
   TextField "Casella di testo_17" at 321,382 size 96x20; Text 'numero di cicli'
   TextField "Casella di testo_18" at 727,60 size 49x17; Text 'SQ_alto'
   TextField "Casella di testo_19" at 725,237 size 60x17; Text 'SQ_basso'
   TextField "Casella di testo_20" at 498,384 size 55x17; Text 'BC_inizio'
   TextField "Casella di testo_21" at 668,383 size 47x17; Text 'BC_fine'
   TextField "Casella di testo_22" at 487,61 size 91x20; Text 'in movimento'
   TextField "Casella di testo_23" at 316,23 size 39x20; Text 'Start'
   Switch "Interruttore_1" at 503,363 size 45x21; CaptionText 'Switch'; TextOff 'OFF'; TextOn 'ON'
      on SwitchOn: SetBit("Blocco_dati_HMI_jog_BC_inizio")
      on SwitchOff: ResetBit("Blocco_dati_HMI_jog_BC_inizio")
   Switch "Interruttore_2" at 674,362 size 45x21; TextOn 'ON'; CaptionText 'Switch'; TextOff 'OFF'
      on SwitchOn: SetBit("Blocco_dati_HMI_jog_BC_fine")
      on SwitchOff: ResetBit("Blocco_dati_HMI_jog_BC_fine")
   Switch "Interruttore_3" at 727,81 size 45x21; TextOn 'ON'; CaptionText 'Switch'; TextOff 'OFF'
      on SwitchOn: SetBit("Blocco_dati_HMI_jog_SQ_alto")
      on SwitchOff: ResetBit("Blocco_dati_HMI_jog_SQ_alto")
   Switch "Interruttore_4" at 728,259 size 45x21; TextOn 'ON'; CaptionText 'Switch'; TextOff 'OFF'
      on SwitchOn: SetBit("Blocco_dati_HMI_jog_SQ_basso")
      on SwitchOff: ResetBit("Blocco_dati_HMI_jog_SQ_basso")
   GraphicIOField "PlotLight_Round_R" at 499,77 size 50x50; PictureOn "PilotLight_Round_R_On_256c"; PictureOff "PilotLight_Round_R_Off_256c"
      ProcessValue <- "Blocco_dati_HMI_Spia organi in movimento"
   GraphicIOField "PlotLight_Round_G" at 685,398 size 30x30; PictureOn "PilotLight_Round_G_On_256c"; PictureOff "PilotLight_Round_G_Off_256c"
      ProcessValue <- "Blocco_dati_HMI_Spia_BC_fine"
   GraphicIOField "PlotLight_Round_G_1" at 515,398 size 30x30; PictureOff "PilotLight_Round_G_Off_256c"; PictureOn "PilotLight_Round_G_On_256c"
      ProcessValue <- "Blocco_dati_HMI_Spia_BC_inizio"
   GraphicIOField "PlotLight_Round_G_2" at 738,280 size 30x30; PictureOff "PilotLight_Round_G_Off_256c"; PictureOn "PilotLight_Round_G_On_256c"
      ProcessValue <- "Blocco_dati_HMI_Spia _SQ_basso"
   GraphicIOField "PlotLight_Round_G_3" at 737,102 size 30x30; PictureOff "PilotLight_Round_G_Off_256c"; PictureOn "PilotLight_Round_G_On_256c"
      ProcessValue <- "Blocco_dati_HMI_Spia_SQ_alto"
   GraphicView "Vista grafica_1" at 653,77 size 53x86; Picture "Mandrino_1"
      VerticalMovement <- "Blocco_dati_HMI_movimento lavorazione"
*)